(* CoDeSys 2.3.9.37 project: Cap5_1.pro *)
(* Libraries: Standard.lib 4.10.05 12:14:46 *)

(* Global variable list: Global_Variables *)
VAR_GLOBAL
 (* Variables de entrada *)
   BotonS : BOOL;
   BotonR : BOOL;
(* Variables de salida *)
   Salida: BOOL;
END_VAR

(* POU PLC_PRG, FBD *)
PROGRAM PLC_PRG
VAR

   MiBiestable : Biestable;

END_VAR
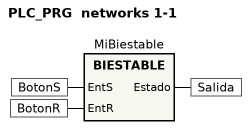
_FBD_ (* Function Block Diagram *)
NETWORK 1
	MiBiestable:BIESTABLE(EntS: BotonS, EntR: BotonR) => Salida
_END_FBD_
(* the same logic as Structured Text *)
(* Network 1 *)
MiBiestable(EntS := BotonS, EntR := BotonR);
Salida := MiBiestable.Estado;
END_PROGRAM

(* POU Biestable, ST *)
FUNCTION_BLOCK Biestable
VAR_INPUT
   EntS : BOOL;
   EntR:BOOL;
END_VAR
VAR_OUTPUT
    Estado : BOOL := FALSE;
END_VAR
VAR
END_VAR
IF (EntS=TRUE ) THEN
   Estado:=TRUE;
ELSE
   IF (EntR=TRUE) THEN
       Estado:=FALSE;
   END_IF
END_IF
END_FUNCTION_BLOCK

(* Visualisation Biestable
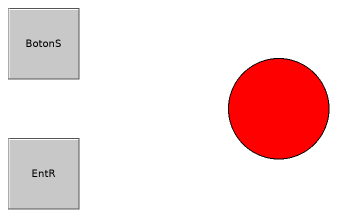
button at (110,80)-(181,151): text "BotonS"; taps BotonS
button at (110,210)-(181,281): text "EntR"; taps BotonR
ellipse at (330,130)-(431,231): alarm colour if Salida
*)
